FUNCTION IsValidImage : BOOL
VAR_INPUT
    Image : ITcVnImage;
END_VAR

IsValidImage := Image <> 0;

END_FUNCTION

(* stored: Version 1.1.0.1, ProductVersion 3.1.4024.13
   POU IsValidImage: Id {4f5abcd5-0122-0350-3fa7-716c6d734fe9}, SpecialFunc None *)
